LIN {X 0,Y 82.833,Z 534.203,A -85,B 0,C 180,E1 -27639.758,E2 -27639.758} C_VEL
LIN {X 0,Y 83.989,Z 533.266,A -85,B 0,C 180,E1 -27644.526,E2 -27644.526} C_VEL
LIN {X 0,Y 85.511,Z 531.952,A -85,B 0,C 180,E1 -27649.181,E2 -27649.181} C_VEL
LIN {X 0,Y 88.778,Z 529.155,A -85,B 0,C 180,E1 -27655.798,E2 -27655.798} C_VEL
LIN {X 0,Y 93.286,Z 525.282,A -85,B 0,C 180,E1 -27661.815,E2 -27661.815} C_VEL
LIN {X 0,Y 98.668,Z 520.245,A -85,B 0,C 180,E1 -27667.247,E2 -27667.247} C_VEL
LIN {X 0,Y 105.001,Z 513.4,A -85,B 0,C 180,E1 -27672.584,E2 -27672.584} C_VEL
LIN {X 0,Y 110.86,Z 506.1,A -85,B 0,C 180,E1 -27676.792,E2 -27676.792} C_VEL
LIN {X 0,Y 116.617,Z 498.037,A -85,B 0,C 180,E1 -27680.194,E2 -27680.194} C_VEL
LIN {X 0,Y 121.989,Z 489.202,A -85,B 0,C 180,E1 -27683.054,E2 -27683.054} C_VEL
LIN {X 0,Y 127.559,Z 478.2,A -85,B 0,C 180,E1 -27685.719,E2 -27685.719} C_VEL
LIN {X 0,Y 128.173,Z 476.919,A -85,B 0,C 180,E1 -27685.963,E2 -27685.963} C_VEL
LIN {X 0,Y 128.999,Z 471.512,A -85,B 0,C 180,E1 -27688.215,E2 -27688.215} C_VEL
LIN {X 0,Y 128.591,Z 466.823,A -85,B 0,C 180,E1 -27690.963,E2 -27690.963} C_VEL
LIN {X 0,Y 127.608,Z 461.168,A -85,B 0,C 180,E1 -27694.732,E2 -27694.732} C_VEL
LIN {X 0,Y 126.153,Z 455.519,A -85,B 0,C 180,E1 -27699.313,E2 -27699.313} C_VEL
LIN {X 0,Y 124.735,Z 451.921,A -85,B 0,C 180,E1 -27703.39,E2 -27703.39} C_VEL
LIN {X 0,Y 123.462,Z 448.563,A -85,B 0,C 180,E1 -27708.09,E2 -27708.09} C_VEL
LIN {X 0,Y 122.428,Z 445.351,A -85,B 0,C 180,E1 -27715.059,E2 -27715.059} C_VEL
LIN {X 0,Y 122.377,Z 444.889,A -85,B 0,C 180,E1 -27720.41,E2 -27720.41} C_VEL
LIN {X 0,Y 122.486,Z 446.263,A -85,B 0,C 180,E1 -27723.288,E2 -27723.288} C_VEL
LIN {X 0,Y 123.15,Z 449.904,A -85,B 0,C 180,E1 -27728.304,E2 -27728.304} C_VEL
LIN {X 0,Y 124.989,Z 457.619,A -85,B 0,C 180,E1 -27735.177,E2 -27735.177} C_VEL
LIN {X 0,Y 126.556,Z 464.817,A -85,B 0,C 180,E1 -27739.778,E2 -27739.778} C_VEL
LIN {X 0,Y 127.843,Z 470.42,A -85,B 0,C 180,E1 -27743.015,E2 -27743.015} C_VEL
LIN {X 0,Y 125.155,Z 484.311,A -85,B 0,C 180,E1 -27746.063,E2 -27746.063} C_VEL
LIN {X 0,Y 123.577,Z 490.066,A -85,B 0,C 180,E1 -27747.393,E2 -27747.393} C_VEL
LIN {X 0,Y 118.187,Z 501.884,A -85,B 0,C 180,E1 -27749.598,E2 -27749.598} C_VEL
LIN {X 0,Y 112.239,Z 512.594,A -85,B 0,C 180,E1 -27752.312,E2 -27752.312} C_VEL
LIN {X 0,Y 106.056,Z 522.326,A -85,B 0,C 180,E1 -27755.749,E2 -27755.749} C_VEL
LIN {X 0,Y 100.298,Z 530.329,A -85,B 0,C 180,E1 -27759.592,E2 -27759.592} C_VEL
LIN {X 0,Y 94.122,Z 538.214,A -85,B 0,C 180,E1 -27764.833,E2 -27764.833} C_VEL
LIN {X 0,Y 88.78,Z 544.608,A -85,B 0,C 180,E1 -27770.722,E2 -27770.722} C_VEL
LIN {X 0,Y 84.577,Z 549.746,A -85,B 0,C 180,E1 -27777.323,E2 -27777.323} C_VEL
LIN {X 0,Y 81.613,Z 553.757,A -85,B 0,C 180,E1 -27784.51,E2 -27784.51} C_VEL
LIN {X 0,Y 80.342,Z 555.873,A -85,B 0,C 180,E1 -27789.532,E2 -27789.532} C_VEL
LIN {X 0,Y 79.565,Z 557.948,A -85,B 0,C 180,E1 -27796.314,E2 -27796.314} C_VEL
LIN {X 0,Y 79.705,Z 559.51,A -85,B 0,C 180,E1 -27804.954,E2 -27804.954} C_VEL
LIN {X 0,Y 80.417,Z 559.877,A -85,B 0,C 180,E1 -27810.012,E2 -27810.012} C_VEL
LIN {X 0,Y 79.813,Z 559.509,A -85,B 0,C 180,E1 -27815.064,E2 -27815.064} C_VEL
LIN {X 0,Y 79.646,Z 558.723,A -85,B 0,C 180,E1 -27820.177,E2 -27820.177} C_VEL
LIN {X 0,Y 79.905,Z 557.516,A -85,B 0,C 180,E1 -27825.312,E2 -27825.312} C_VEL
LIN {X 0,Y 81.437,Z 554.888,A -85,B 0,C 180,E1 -27832.864,E2 -27832.864} C_VEL
LIN {X 0,Y 84.334,Z 551.27,A -85,B 0,C 180,E1 -27840.013,E2 -27840.013} C_VEL
LIN {X 0,Y 89.332,Z 545.786,A -85,B 0,C 180,E1 -27847.457,E2 -27847.457} C_VEL
LIN {X 0,Y 89.839,Z 545.307,A -85,B 0,C 180,E1 -27847.979,E2 -27847.979} C_VEL
LIN {X 0,Y 101.006,Z 544.866,A -85,B 0,C 180,E1 -27859.954,E2 -27859.954} C_VEL
LIN {X 0,Y 105.346,Z 544.467,A -85,B 0,C 180,E1 -27863.102,E2 -27863.102} C_VEL
LIN {X 0,Y 96.759,Z 538.849,A -85,B 0,C 180,E1 -27869.442,E2 -27869.442} C_VEL
LIN {X 0,Y 88.329,Z 530.261,A -85,B 0,C 180,E1 -27879.022,E2 -27879.022} C_VEL
LIN {X 0,Y 83.096,Z 520.814,A -85,B 0,C 180,E1 -27889.032,E2 -27889.032} C_VEL
LIN {X 0,Y 82.33,Z 518.793,A -85,B 0,C 180,E1 -27891.411,E2 -27891.411} C_VEL
LIN {X 0,Y 81.635,Z 518.051,A -85,B 0,C 180,E1 -27895.063,E2 -27895.063} C_VEL
LIN {X 0,Y 82.102,Z 516.286,A -85,B 0,C 180,E1 -27900.002,E2 -27900.002} C_VEL
LIN {X 0,Y 82.708,Z 514.93,A -85,B 0,C 180,E1 -27904.876,E2 -27904.876} C_VEL
LIN {X 0,Y 84.487,Z 513.029,A -85,B 0,C 180,E1 -27909.579,E2 -27909.579} C_VEL
LIN {X 0,Y 88.142,Z 510.312,A -85,B 0,C 180,E1 -27916.865,E2 -27916.865} C_VEL
LIN {X 0,Y 96.42,Z 505.521,A -85,B 0,C 180,E1 -27925.936,E2 -27925.936} C_VEL
LIN {X 0,Y 105.323,Z 501.018,A -85,B 0,C 180,E1 -27932.266,E2 -27932.266} C_VEL
LIN {X 0,Y 110.649,Z 498.102,A -85,B 0,C 180,E1 -27934.867,E2 -27934.867} C_VEL
LIN {X 0,Y 114.44,Z 496.301,A -85,B 0,C 180,E1 -27936.743,E2 -27936.743} C_VEL
LIN {X 0,Y 114.902,Z 496.45,A -85,B 0,C 180,E1 -27937.289,E2 -27937.289} C_VEL
LIN {X 0,Y 114.491,Z 497.858,A -85,B 0,C 180,E1 -27938.218,E2 -27938.218} C_VEL
LIN {X 0,Y 112.735,Z 500.446,A -85,B 0,C 180,E1 -27939.209,E2 -27939.209} C_VEL
LIN {X 0,Y 105.09,Z 508.492,A -85,B 0,C 180,E1 -27941.444,E2 -27941.444} C_VEL
LIN {X 0,Y 103.107,Z 510.663,A -85,B 0,C 180,E1 -27942.499,E2 -27942.499} C_VEL
LIN {X 0,Y 96.352,Z 518.081,A -85,B 0,C 180,E1 -27947.556,E2 -27947.556} C_VEL
LIN {X 0,Y 89.384,Z 524.598,A -85,B 0,C 180,E1 -27953.851,E2 -27953.851} C_VEL
LIN {X 0,Y 84.032,Z 528.908,A -85,B 0,C 180,E1 -27959.868,E2 -27959.868} C_VEL
LIN {X 0,Y 81.236,Z 531.13,A -85,B 0,C 180,E1 -27964.357,E2 -27964.357} C_VEL
LIN {X 0,Y 78.937,Z 532.932,A -85,B 0,C 180,E1 -27969.124,E2 -27969.124} C_VEL
LIN {X 0,Y 77.222,Z 534.283,A -85,B 0,C 180,E1 -27974.142,E2 -27974.142} C_VEL
LIN {X 0,Y 75.944,Z 535.235,A -85,B 0,C 180,E1 -27979.321,E2 -27979.321} C_VEL
LIN {X 0,Y 74.808,Z 536.056,A -85,B 0,C 180,E1 -27989.987,E2 -27989.987} C_VEL
LIN {X 0,Y 75.939,Z 535.278,A -85,B 0,C 180,E1 -28000.653,E2 -28000.653} C_VEL
LIN {X 0,Y 77.211,Z 534.343,A -85,B 0,C 180,E1 -28005.834,E2 -28005.834} C_VEL
LIN {X 0,Y 78.913,Z 533.029,A -85,B 0,C 180,E1 -28010.856,E2 -28010.856} C_VEL
LIN {X 0,Y 82.515,Z 530.23,A -85,B 0,C 180,E1 -28017.92,E2 -28017.92} C_VEL
LIN {X 0,Y 87.401,Z 526.356,A -85,B 0,C 180,E1 -28024.24,E2 -28024.24} C_VEL
LIN {X 0,Y 93.181,Z 521.318,A -85,B 0,C 180,E1 -28029.859,E2 -28029.859} C_VEL
LIN {X 0,Y 100.066,Z 514.349,A -85,B 0,C 180,E1 -28035.383,E2 -28035.383} C_VEL
LIN {X 0,Y 106.178,Z 507.169,A -85,B 0,C 180,E1 -28039.554,E2 -28039.554} C_VEL
LIN {X 0,Y 112.253,Z 499.104,A -85,B 0,C 180,E1 -28042.948,E2 -28042.948} C_VEL
LIN {X 0,Y 117.905,Z 490.264,A -85,B 0,C 180,E1 -28045.78,E2 -28045.78} C_VEL
LIN {X 0,Y 123.741,Z 479.256,A -85,B 0,C 180,E1 -28048.406,E2 -28048.406} C_VEL
LIN {X 0,Y 124.423,Z 476.66,A -85,B 0,C 180,E1 -28049.444,E2 -28049.444} C_VEL
LIN {X 0,Y 124.623,Z 473.65,A -85,B 0,C 180,E1 -28051.107,E2 -28051.107} C_VEL
LIN {X 0,Y 124.263,Z 468.236,A -85,B 0,C 180,E1 -28054.791,E2 -28054.791} C_VEL
LIN {X 0,Y 123.587,Z 463.882,A -85,B 0,C 180,E1 -28058.306,E2 -28058.306} C_VEL
LIN {X 0,Y 122.813,Z 460.538,A -85,B 0,C 180,E1 -28061.654,E2 -28061.654} C_VEL
LIN {X 0,Y 122.045,Z 457.833,A -85,B 0,C 180,E1 -28064.98,E2 -28064.98} C_VEL
LIN {X 0,Y 121.32,Z 455.06,A -85,B 0,C 180,E1 -28069.147,E2 -28069.147} C_VEL
LIN {X 0,Y 120.821,Z 452.168,A -85,B 0,C 180,E1 -28075.829,E2 -28075.829} C_VEL
LIN {X 0,Y 120.907,Z 451.946,A -85,B 0,C 180,E1 -28080.415,E2 -28080.415} C_VEL
LIN {X 0,Y 120.951,Z 453.628,A -85,B 0,C 180,E1 -28083.538,E2 -28083.538} C_VEL
LIN {X 0,Y 121.287,Z 456.551,A -85,B 0,C 180,E1 -28087.385,E2 -28087.385} C_VEL
LIN {X 0,Y 122.41,Z 463.559,A -85,B 0,C 180,E1 -28093.804,E2 -28093.804} C_VEL
LIN {X 0,Y 123.355,Z 470.169,A -85,B 0,C 180,E1 -28098.216,E2 -28098.216} C_VEL
LIN {X 0,Y 124.012,Z 474.29,A -85,B 0,C 180,E1 -28100.744,E2 -28100.744} C_VEL
LIN {X 0,Y 120.797,Z 487.152,A -85,B 0,C 180,E1 -28103.743,E2 -28103.743} C_VEL
LIN {X 0,Y 119.72,Z 490.608,A -85,B 0,C 180,E1 -28104.596,E2 -28104.596} C_VEL
LIN {X 0,Y 114.096,Z 502.097,A -85,B 0,C 180,E1 -28106.748,E2 -28106.748} C_VEL
LIN {X 0,Y 107.866,Z 512.581,A -85,B 0,C 180,E1 -28109.393,E2 -28109.393} C_VEL
LIN {X 0,Y 101.992,Z 521.223,A -85,B 0,C 180,E1 -28112.443,E2 -28112.443} C_VEL
LIN {X 0,Y 94.669,Z 530.629,A -85,B 0,C 180,E1 -28117.074,E2 -28117.074} C_VEL
LIN {X 0,Y 88.108,Z 538.272,A -85,B 0,C 180,E1 -28122.471,E2 -28122.471} C_VEL
LIN {X 0,Y 81.565,Z 545.347,A -85,B 0,C 180,E1 -28129.758,E2 -28129.758} C_VEL
LIN {X 0,Y 77.256,Z 550.092,A -85,B 0,C 180,E1 -28136.935,E2 -28136.935} C_VEL
LIN {X 0,Y 74.301,Z 553.756,A -85,B 0,C 180,E1 -28144.823,E2 -28144.823} C_VEL
LIN {X 0,Y 72.561,Z 556.992,A -85,B 0,C 180,E1 -28155.588,E2 -28155.588} C_VEL
LIN {X 0,Y 72.613,Z 558.418,A -85,B 0,C 180,E1 -28164.459,E2 -28164.459} C_VEL
LIN {X 0,Y 73.336,Z 558.791,A -85,B 0,C 180,E1 -28170.013,E2 -28170.013} C_VEL
LIN {X 0,Y 72.723,Z 558.417,A -85,B 0,C 180,E1 -28175.559,E2 -28175.559} C_VEL
LIN {X 0,Y 72.838,Z 556.784,A -85,B 0,C 180,E1 -28185.237,E2 -28185.237} C_VEL
LIN {X 0,Y 74.855,Z 553.783,A -85,B 0,C 180,E1 -28195.006,E2 -28195.006} C_VEL
LIN {X 0,Y 78.192,Z 550.167,A -85,B 0,C 180,E1 -28202.649,E2 -28202.649} C_VEL
LIN {X 0,Y 82.904,Z 545.488,A -85,B 0,C 180,E1 -28209.493,E2 -28209.493} C_VEL
LIN {X 0,Y 86.143,Z 542.479,A -85,B 0,C 180,E1 -28212.874,E2 -28212.874} C_VEL
LIN {X 0,Y 95.313,Z 542.275,A -85,B 0,C 180,E1 -28221.931,E2 -28221.931} C_VEL
LIN {X 0,Y 96.208,Z 542.082,A -85,B 0,C 180,E1 -28222.918,E2 -28222.918} C_VEL
LIN {X 0,Y 86.816,Z 534.865,A -85,B 0,C 180,E1 -28230.943,E2 -28230.943} C_VEL
LIN {X 0,Y 79.323,Z 525.924,A -85,B 0,C 180,E1 -28241.268,E2 -28241.268} C_VEL
LIN {X 0,Y 77.81,Z 525.42,A -85,B 0,C 180,E1 -28244.28,E2 -28244.28} C_VEL
LIN {X 0,Y 78.095,Z 518.652,A -85,B 0,C 180,E1 -28268.064,E2 -28268.064} C_VEL
LIN {X 0,Y 84.543,Z 514.175,A -85,B 0,C 180,E1 -28280.207,E2 -28280.207} C_VEL
LIN {X 0,Y 93.773,Z 509.487,A -85,B 0,C 180,E1 -28289.156,E2 -28289.156} C_VEL
LIN {X 0,Y 100.734,Z 506.327,A -85,B 0,C 180,E1 -28293.929,E2 -28293.929} C_VEL
LIN {X 0,Y 108.996,Z 502.319,A -85,B 0,C 180,E1 -28297.779,E2 -28297.779} C_VEL
LIN {X 0,Y 108.664,Z 503.744,A -85,B 0,C 180,E1 -28299.081,E2 -28299.081} C_VEL
LIN {X 0,Y 103.107,Z 510.663,A -85,B 0,C 180,E1 -28302.499,E2 -28302.499} C_VEL
LIN {X 0,Y 99.686,Z 514.194,A -85,B 0,C 180,E1 -28304.373,E2 -28304.373} C_VEL
LIN {X 0,Y 92.734,Z 519.7,A -85,B 0,C 180,E1 -28307.025,E2 -28307.025} C_VEL
LIN {X 0,Y 85.549,Z 524.579,A -85,B 0,C 180,E1 -28310.147,E2 -28310.147} C_VEL
LIN {X 0,Y 81.903,Z 527.126,A -85,B 0,C 180,E1 -28312.816,E2 -28312.816} C_VEL
LIN {X 0,Y 76.426,Z 531.174,A -85,B 0,C 180,E1 -28319.603,E2 -28319.603} C_VEL
LIN {X 0,Y 72.42,Z 534.01,A -85,B 0,C 180,E1 -28327.145,E2 -28327.145} C_VEL
LIN {X 0,Y 70.492,Z 535.361,A -85,B 0,C 180,E1 -28332.583,E2 -28332.583} C_VEL
LIN {X 0,Y 69.07,Z 536.31,A -85,B 0,C 180,E1 -28338.244,E2 -28338.244} C_VEL
LIN {X 0,Y 67.791,Z 537.133,A -85,B 0,C 180,E1 -28349.986,E2 -28349.986} C_VEL
LIN {X 0,Y 69.064,Z 536.353,A -85,B 0,C 180,E1 -28361.728,E2 -28361.728} C_VEL
LIN {X 0,Y 70.48,Z 535.42,A -85,B 0,C 180,E1 -28367.392,E2 -28367.392} C_VEL
LIN {X 0,Y 72.395,Z 534.105,A -85,B 0,C 180,E1 -28372.834,E2 -28372.834} C_VEL
LIN {X 0,Y 76.384,Z 531.306,A -85,B 0,C 180,E1 -28380.386,E2 -28380.386} C_VEL
LIN {X 0,Y 81.695,Z 527.431,A -85,B 0,C 180,E1 -28387.011,E2 -28387.011} C_VEL
LIN {X 0,Y 87.911,Z 522.39,A -85,B 0,C 180,E1 -28392.79,E2 -28392.79} C_VEL
LIN {X 0,Y 95.307,Z 515.38,A -85,B 0,C 180,E1 -28398.418,E2 -28398.418} C_VEL
LIN {X 0,Y 101.77,Z 508.237,A -85,B 0,C 180,E1 -28402.558,E2 -28402.558} C_VEL
LIN {X 0,Y 108.174,Z 500.169,A -85,B 0,C 180,E1 -28405.913,E2 -28405.913} C_VEL
LIN {X 0,Y 114.108,Z 491.325,A -85,B 0,C 180,E1 -28408.694,E2 -28408.694} C_VEL
LIN {X 0,Y 119.658,Z 481.481,A -85,B 0,C 180,E1 -28410.991,E2 -28410.991} C_VEL
LIN {X 0,Y 120.04,Z 480.367,A -85,B 0,C 180,E1 -28411.408,E2 -28411.408} C_VEL
LIN {X 0,Y 120.371,Z 477.712,A -85,B 0,C 180,E1 -28413.038,E2 -28413.038} C_VEL
LIN {X 0,Y 120.385,Z 472.643,A -85,B 0,C 180,E1 -28416.792,E2 -28416.792} C_VEL
LIN {X 0,Y 119.988,Z 467.797,A -85,B 0,C 180,E1 -28421.206,E2 -28421.206} C_VEL
LIN {X 0,Y 119.505,Z 464.937,A -85,B 0,C 180,E1 -28424.653,E2 -28424.653} C_VEL
LIN {X 0,Y 118.986,Z 461.601,A -85,B 0,C 180,E1 -28429.792,E2 -28429.792} C_VEL
LIN {X 0,Y 118.898,Z 458.901,A -85,B 0,C 180,E1 -28436.61,E2 -28436.61} C_VEL
LIN {X 0,Y 119.048,Z 458.863,A -85,B 0,C 180,E1 -28440.421,E2 -28440.421} C_VEL
LIN {X 0,Y 119.078,Z 462.44,A -85,B 0,C 180,E1 -28445.821,E2 -28445.821} C_VEL
LIN {X 0,Y 119.52,Z 468.513,A -85,B 0,C 180,E1 -28451.739,E2 -28451.739} C_VEL
LIN {X 0,Y 119.946,Z 474.653,A -85,B 0,C 180,E1 -28456.158,E2 -28456.158} C_VEL
LIN {X 0,Y 120.179,Z 478.222,A -85,B 0,C 180,E1 -28458.407,E2 -28458.407} C_VEL
LIN {X 0,Y 116.094,Z 491.174,A -85,B 0,C 180,E1 -28461.605,E2 -28461.605} C_VEL
LIN {X 0,Y 110.309,Z 502.311,A -85,B 0,C 180,E1 -28463.697,E2 -28463.697} C_VEL
LIN {X 0,Y 103.803,Z 512.522,A -85,B 0,C 180,E1 -28466.245,E2 -28466.245} C_VEL
LIN {X 0,Y 96.945,Z 521.809,A -85,B 0,C 180,E1 -28469.572,E2 -28469.572} C_VEL
LIN {X 0,Y 89.242,Z 530.924,A -85,B 0,C 180,E1 -28474.241,E2 -28474.241} C_VEL
LIN {X 0,Y 82.254,Z 538.296,A -85,B 0,C 180,E1 -28479.757,E2 -28479.757} C_VEL
LIN {X 0,Y 76.15,Z 544.232,A -85,B 0,C 180,E1 -28486.215,E2 -28486.215} C_VEL
LIN {X 0,Y 71.271,Z 548.978,A -85,B 0,C 180,E1 -28493.743,E2 -28493.743} C_VEL
LIN {X 0,Y 67.8,Z 552.643,A -85,B 0,C 180,E1 -28502.212,E2 -28502.212} C_VEL
LIN {X 0,Y 65.571,Z 556.036,A -85,B 0,C 180,E1 -28514.708,E2 -28514.708} C_VEL
LIN {X 0,Y 65.526,Z 557.325,A -85,B 0,C 180,E1 -28523.858,E2 -28523.858} C_VEL
LIN {X 0,Y 66.253,Z 557.704,A -85,B 0,C 180,E1 -28530.015,E2 -28530.015} C_VEL
LIN {X 0,Y 65.636,Z 557.323,A -85,B 0,C 180,E1 -28536.162,E2 -28536.162} C_VEL
LIN {X 0,Y 65.857,Z 555.831,A -85,B 0,C 180,E1 -28546.177,E2 -28546.177} C_VEL
LIN {X 0,Y 68.404,Z 552.679,A -85,B 0,C 180,E1 -28557.554,E2 -28557.554} C_VEL
LIN {X 0,Y 72.253,Z 549.065,A -85,B 0,C 180,E1 -28565.721,E2 -28565.721} C_VEL
LIN {X 0,Y 77.499,Z 544.386,A -85,B 0,C 180,E1 -28572.87,E2 -28572.87} C_VEL
LIN {X 0,Y 83.213,Z 539.471,A -85,B 0,C 180,E1 -28578.113,E2 -28578.113} C_VEL
LIN {X 0,Y 83.961,Z 539.481,A -85,B 0,C 180,E1 -28578.898,E2 -28578.898} C_VEL
LIN {X 0,Y 86.779,Z 538.866,A -85,B 0,C 180,E1 -28583.025,E2 -28583.025} C_VEL
LIN {X 0,Y 79.255,Z 532.702,A -85,B 0,C 180,E1 -28590.082,E2 -28590.082} C_VEL
LIN {X 0,Y 77.027,Z 532.131,A -85,B 0,C 180,E1 -28592.86,E2 -28592.86} C_VEL
LIN {X 0,Y 70.369,Z 526.801,A -85,B 0,C 180,E1 -28614.27,E2 -28614.27} C_VEL
LIN {X 0,Y 73.252,Z 522.271,A -85,B 0,C 180,E1 -28631.065,E2 -28631.065} C_VEL
LIN {X 0,Y 82.345,Z 517.135,A -85,B 0,C 180,E1 -28645.263,E2 -28645.263} C_VEL
LIN {X 0,Y 98.671,Z 510.136,A -85,B 0,C 180,E1 -28657.201,E2 -28657.201} C_VEL
LIN {X 0,Y 100.317,Z 509.415,A -85,B 0,C 180,E1 -28657.976,E2 -28657.976} C_VEL
LIN {X 0,Y 98.411,Z 511.85,A -85,B 0,C 180,E1 -28659.561,E2 -28659.561} C_VEL
LIN {X 0,Y 91.299,Z 519.157,A -85,B 0,C 180,E1 -28664.585,E2 -28664.585} C_VEL
LIN {X 0,Y 83.818,Z 525.675,A -85,B 0,C 180,E1 -28671.02,E2 -28671.02} C_VEL
LIN {X 0,Y 81.903,Z 527.126,A -85,B 0,C 180,E1 -28672.816,E2 -28672.816} C_VEL
LIN {X 0,Y 78.412,Z 529.488,A -85,B 0,C 180,E1 -28675.791,E2 -28675.791} C_VEL
LIN {X 0,Y 71.806,Z 532.945,A -85,B 0,C 180,E1 -28680.787,E2 -28680.787} C_VEL
LIN {X 0,Y 65.833,Z 535.556,A -85,B 0,C 180,E1 -28686.962,E2 -28686.962} C_VEL
LIN {X 0,Y 63.52,Z 536.591,A -85,B 0,C 180,E1 -28691.669,E2 -28691.669} C_VEL
LIN {X 0,Y 61.144,Z 537.985,A -85,B 0,C 180,E1 -28703.384,E2 -28703.384} C_VEL
LIN {X 0,Y 60.774,Z 538.21,A -85,B 0,C 180,E1 -28709.984,E2 -28709.984} C_VEL
LIN {X 0,Y 62.216,Z 537.428,A -85,B 0,C 180,E1 -28723.041,E2 -28723.041} C_VEL
LIN {X 0,Y 63.812,Z 536.497,A -85,B 0,C 180,E1 -28729.277,E2 -28729.277} C_VEL
LIN {X 0,Y 65.98,Z 535.182,A -85,B 0,C 180,E1 -28735.201,E2 -28735.201} C_VEL
LIN {X 0,Y 70.418,Z 532.381,A -85,B 0,C 180,E1 -28743.275,E2 -28743.275} C_VEL
LIN {X 0,Y 76.209,Z 528.505,A -85,B 0,C 180,E1 -28750.188,E2 -28750.188} C_VEL
LIN {X 0,Y 82.901,Z 523.463,A -85,B 0,C 180,E1 -28756.085,E2 -28756.085} C_VEL
LIN {X 0,Y 90.088,Z 517.141,A -85,B 0,C 180,E1 -28761.253,E2 -28761.253} C_VEL
LIN {X 0,Y 97.666,Z 509.306,A -85,B 0,C 180,E1 -28765.827,E2 -28765.827} C_VEL
LIN {X 0,Y 104.404,Z 501.235,A -85,B 0,C 180,E1 -28769.102,E2 -28769.102} C_VEL
LIN {X 0,Y 110.624,Z 492.388,A -85,B 0,C 180,E1 -28771.801,E2 -28771.801} C_VEL
LIN {X 0,Y 115.596,Z 484.106,A -85,B 0,C 180,E1 -28773.687,E2 -28773.687} C_VEL
LIN {X 0,Y 116.05,Z 482.696,A -85,B 0,C 180,E1 -28774.358,E2 -28774.358} C_VEL
LIN {X 0,Y 116.5,Z 478.229,A -85,B 0,C 180,E1 -28777.847,E2 -28777.847} C_VEL
LIN {X 0,Y 116.581,Z 473.471,A -85,B 0,C 180,E1 -28782.456,E2 -28782.456} C_VEL
LIN {X 0,Y 116.406,Z 470.759,A -85,B 0,C 180,E1 -28786.024,E2 -28786.024} C_VEL
LIN {X 0,Y 116.332,Z 468.587,A -85,B 0,C 180,E1 -28789.557,E2 -28789.557} C_VEL
LIN {X 0,Y 116.58,Z 465.75,A -85,B 0,C 180,E1 -28796.542,E2 -28796.542} C_VEL
LIN {X 0,Y 116.788,Z 465.606,A -85,B 0,C 180,E1 -28799.999,E2 -28799.999} C_VEL
LIN {X 0,Y 116.633,Z 467.681,A -85,B 0,C 180,E1 -28803.453,E2 -28803.453} C_VEL
LIN {X 0,Y 116.441,Z 472.562,A -85,B 0,C 180,E1 -28808.677,E2 -28808.677} C_VEL
LIN {X 0,Y 116.481,Z 475.544,A -85,B 0,C 180,E1 -28811.307,E2 -28811.307} C_VEL
LIN {X 0,Y 116.408,Z 481.703,A -85,B 0,C 180,E1 -28815.761,E2 -28815.761} C_VEL
LIN {X 0,Y 112.784,Z 491.752,A -85,B 0,C 180,E1 -28818.416,E2 -28818.416} C_VEL
LIN {X 0,Y 108.375,Z 499.921,A -85,B 0,C 180,E1 -28819.926,E2 -28819.926} C_VEL
LIN {X 0,Y 101.567,Z 510.394,A -85,B 0,C 180,E1 -28822.285,E2 -28822.285} C_VEL
LIN {X 0,Y 95.001,Z 519.017,A -85,B 0,C 180,E1 -28825.038,E2 -28825.038} C_VEL
LIN {X 0,Y 87.092,Z 527.975,A -85,B 0,C 180,E1 -28829.13,E2 -28829.13} C_VEL
LIN {X 0,Y 79.014,Z 536.048,A -85,B 0,C 180,E1 -28834.662,E2 -28834.662} C_VEL
LIN {X 0,Y 73.201,Z 541.269,A -85,B 0,C 180,E1 -28839.841,E2 -28839.841} C_VEL
LIN {X 0,Y 67.641,Z 546.072,A -85,B 0,C 180,E1 -28846.658,E2 -28846.658} C_VEL
LIN {X 0,Y 62.646,Z 550.417,A -85,B 0,C 180,E1 -28855.9,E2 -28855.9} C_VEL
LIN {X 0,Y 60.48,Z 552.545,A -85,B 0,C 180,E1 -28862.321,E2 -28862.321} C_VEL
LIN {X 0,Y 58.573,Z 555.078,A -85,B 0,C 180,E1 -28873.711,E2 -28873.711} C_VEL
LIN {X 0,Y 58.443,Z 556.231,A -85,B 0,C 180,E1 -28883.11,E2 -28883.11} C_VEL
LIN {X 0,Y 59.169,Z 556.617,A -85,B 0,C 180,E1 -28890.017,E2 -28890.017} C_VEL
LIN {X 0,Y 58.559,Z 556.23,A -85,B 0,C 180,E1 -28896.91,E2 -28896.91} C_VEL
LIN {X 0,Y 58.912,Z 554.871,A -85,B 0,C 180,E1 -28907.385,E2 -28907.385} C_VEL
LIN {X 0,Y 62.135,Z 551.578,A -85,B 0,C 180,E1 -28920.614,E2 -28920.614} C_VEL
LIN {X 0,Y 66.552,Z 547.963,A -85,B 0,C 180,E1 -28929.335,E2 -28929.335} C_VEL
LIN {X 0,Y 73.249,Z 542.645,A -85,B 0,C 180,E1 -28937.532,E2 -28937.532} C_VEL
LIN {X 0,Y 76.668,Z 539.855,A -85,B 0,C 180,E1 -28940.555,E2 -28940.555} C_VEL
LIN {X 0,Y 78.011,Z 537.963,A -85,B 0,C 180,E1 -28942.781,E2 -28942.781} C_VEL
LIN {X 0,Y 65.096,Z 532.054,A -85,B 0,C 180,E1 -28967.533,E2 -28967.533} C_VEL
LIN {X 0,Y 67.36,Z 526.292,A -85,B 0,C 180,E1 -28992.047,E2 -28992.047} C_VEL
LIN {X 0,Y 76.977,Z 521.399,A -85,B 0,C 180,E1 -29007.164,E2 -29007.164} C_VEL
LIN {X 0,Y 91.291,Z 515.788,A -85,B 0,C 180,E1 -29018.018,E2 -29018.018} C_VEL
LIN {X 0,Y 85.337,Z 521.292,A -85,B 0,C 180,E1 -29022.15,E2 -29022.15} C_VEL
LIN {X 0,Y 78.486,Z 526.752,A -85,B 0,C 180,E1 -29027.795,E2 -29027.795} C_VEL
LIN {X 0,Y 72.239,Z 531.062,A -85,B 0,C 180,E1 -29034.271,E2 -29034.271} C_VEL
LIN {X 0,Y 68.886,Z 533.279,A -85,B 0,C 180,E1 -29039.313,E2 -29039.313} C_VEL
LIN {X 0,Y 66.008,Z 535.088,A -85,B 0,C 180,E1 -29044.777,E2 -29044.777} C_VEL
LIN {X 0,Y 63.52,Z 536.591,A -85,B 0,C 180,E1 -29051.669,E2 -29051.669} C_VEL
LIN {X 0,Y 61.538,Z 537.505,A -85,B 0,C 180,E1 -29056.717,E2 -29056.717} C_VEL
LIN {X 0,Y 57.434,Z 538.649,A -85,B 0,C 180,E1 -29065.364,E2 -29065.364} C_VEL
LIN {X 0,Y 54.933,Z 539.062,A -85,B 0,C 180,E1 -29073.076,E2 -29073.076} C_VEL
LIN {X 0,Y 54.475,Z 538.96,A -85,B 0,C 180,E1 -29079.272,E2 -29079.272} C_VEL
LIN {X 0,Y 54.718,Z 538.777,A -85,B 0,C 180,E1 -29081.326,E2 -29081.326} C_VEL
LIN {X 0,Y 57.229,Z 537.575,A -85,B 0,C 180,E1 -29091.599,E2 -29091.599} C_VEL
LIN {X 0,Y 59.702,Z 536.258,A -85,B 0,C 180,E1 -29098.072,E2 -29098.072} C_VEL
LIN {X 0,Y 64.665,Z 533.456,A -85,B 0,C 180,E1 -29106.69,E2 -29106.69} C_VEL
LIN {X 0,Y 70.993,Z 529.579,A -85,B 0,C 180,E1 -29113.845,E2 -29113.845} C_VEL
LIN {X 0,Y 78.199,Z 524.535,A -85,B 0,C 180,E1 -29119.79,E2 -29119.79} C_VEL
LIN {X 0,Y 85.876,Z 518.211,A -85,B 0,C 180,E1 -29124.902,E2 -29124.902} C_VEL
LIN {X 0,Y 93.903,Z 510.375,A -85,B 0,C 180,E1 -29129.372,E2 -29129.372} C_VEL
LIN {X 0,Y 100.98,Z 502.302,A -85,B 0,C 180,E1 -29132.522,E2 -29132.522} C_VEL
LIN {X 0,Y 107.487,Z 493.449,A -85,B 0,C 180,E1 -29135.098,E2 -29135.098} C_VEL
LIN {X 0,Y 111.888,Z 486.448,A -85,B 0,C 180,E1 -29136.64,E2 -29136.64} C_VEL
LIN {X 0,Y 112.698,Z 481.88,A -85,B 0,C 180,E1 -29140.687,E2 -29140.687} C_VEL
LIN {X 0,Y 113.024,Z 478.571,A -85,B 0,C 180,E1 -29144.393,E2 -29144.393} C_VEL
LIN {X 0,Y 113.205,Z 475.442,A -85,B 0,C 180,E1 -29149.265,E2 -29149.265} C_VEL
LIN {X 0,Y 113.439,Z 473.727,A -85,B 0,C 180,E1 -29152.881,E2 -29152.881} C_VEL
LIN {X 0,Y 113.826,Z 472.462,A -85,B 0,C 180,E1 -29156.459,E2 -29156.459} C_VEL
LIN {X 0,Y 114.09,Z 472.444,A -85,B 0,C 180,E1 -29159.999,E2 -29159.999} C_VEL
LIN {X 0,Y 113.71,Z 474.81,A -85,B 0,C 180,E1 -29163.542,E2 -29163.542} C_VEL
LIN {X 0,Y 113.257,Z 479.744,A -85,B 0,C 180,E1 -29168.743,E2 -29168.743} C_VEL
LIN {X 0,Y 112.712,Z 485.221,A -85,B 0,C 180,E1 -29173.062,E2 -29173.062} C_VEL
LIN {X 0,Y 110.986,Z 489.615,A -85,B 0,C 180,E1 -29174.346,E2 -29174.346} C_VEL
LIN {X 0,Y 108.9,Z 494.111,A -85,B 0,C 180,E1 -29175.479,E2 -29175.479} C_VEL
LIN {X 0,Y 102.19,Z 504.934,A -85,B 0,C 180,E1 -29177.437,E2 -29177.437} C_VEL
LIN {X 0,Y 95.19,Z 514.272,A -85,B 0,C 180,E1 -29179.754,E2 -29179.754} C_VEL
LIN {X 0,Y 86.251,Z 524.392,A -85,B 0,C 180,E1 -29183.585,E2 -29183.585} C_VEL
LIN {X 0,Y 77.787,Z 532.589,A -85,B 0,C 180,E1 -29188.278,E2 -29188.278} C_VEL
LIN {X 0,Y 71.253,Z 538.197,A -85,B 0,C 180,E1 -29193.057,E2 -29193.057} C_VEL
LIN {X 0,Y 64.203,Z 543.735,A -85,B 0,C 180,E1 -29200.006,E2 -29200.006} C_VEL
LIN {X 0,Y 58.399,Z 548.11,A -85,B 0,C 180,E1 -29208.579,E2 -29208.579} C_VEL
LIN {X 0,Y 54.142,Z 551.429,A -85,B 0,C 180,E1 -29218.742,E2 -29218.742} C_VEL
LIN {X 0,Y 51.604,Z 554.096,A -85,B 0,C 180,E1 -29232.417,E2 -29232.417} C_VEL
LIN {X 0,Y 51.369,Z 555.137,A -85,B 0,C 180,E1 -29242.156,E2 -29242.156} C_VEL
LIN {X 0,Y 52.051,Z 555.524,A -85,B 0,C 180,E1 -29250.019,E2 -29250.019} C_VEL
LIN {X 0,Y 51.491,Z 555.136,A -85,B 0,C 180,E1 -29257.864,E2 -29257.864} C_VEL
LIN {X 0,Y 51.994,Z 553.913,A -85,B 0,C 180,E1 -29268.89,E2 -29268.89} C_VEL
LIN {X 0,Y 56.087,Z 550.478,A -85,B 0,C 180,E1 -29284.345,E2 -29284.345} C_VEL
LIN {X 0,Y 61.165,Z 546.86,A -85,B 0,C 180,E1 -29293.604,E2 -29293.604} C_VEL
LIN {X 0,Y 68.125,Z 541.92,A -85,B 0,C 180,E1 -29301.479,E2 -29301.479} C_VEL
LIN {X 0,Y 69.412,Z 540.962,A -85,B 0,C 180,E1 -29302.594,E2 -29302.594} C_VEL
LIN {X 0,Y 67.164,Z 539.563,A -85,B 0,C 180,E1 -29306.861,E2 -29306.861} C_VEL
LIN {X 0,Y 58.185,Z 534.233,A -85,B 0,C 180,E1 -29333.065,E2 -29333.065} C_VEL
LIN {X 0,Y 61.303,Z 529.964,A -85,B 0,C 180,E1 -29353.258,E2 -29353.258} C_VEL
LIN {X 0,Y 71.504,Z 525.253,A -85,B 0,C 180,E1 -29369.438,E2 -29369.438} C_VEL
LIN {X 0,Y 81.182,Z 521.723,A -85,B 0,C 180,E1 -29377.303,E2 -29377.303} C_VEL
LIN {X 0,Y 80.798,Z 522.368,A -85,B 0,C 180,E1 -29378.46,E2 -29378.46} C_VEL
LIN {X 0,Y 73.438,Z 527.829,A -85,B 0,C 180,E1 -29384.113,E2 -29384.113} C_VEL
LIN {X 0,Y 66.669,Z 532.139,A -85,B 0,C 180,E1 -29390.747,E2 -29390.747} C_VEL
LIN {X 0,Y 62.963,Z 534.354,A -85,B 0,C 180,E1 -29396.057,E2 -29396.057} C_VEL
LIN {X 0,Y 59.733,Z 536.165,A -85,B 0,C 180,E1 -29401.907,E2 -29401.907} C_VEL
LIN {X 0,Y 56.828,Z 537.7,A -85,B 0,C 180,E1 -29409.669,E2 -29409.669} C_VEL
LIN {X 0,Y 54.18,Z 539.062,A -85,B 0,C 180,E1 -29422.529,E2 -29422.529} C_VEL
LIN {X 0,Y 53.757,Z 539.286,A -85,B 0,C 180,E1 -29429.982,E2 -29429.982} C_VEL
LIN {X 0,Y 54.718,Z 538.777,A -85,B 0,C 180,E1 -29441.326,E2 -29441.326} C_VEL
LIN {X 0,Y 55.215,Z 538.49,A -85,B 0,C 180,E1 -29445.384,E2 -29445.384} C_VEL
LIN {X 0,Y 55.541,Z 537.745,A -85,B 0,C 180,E1 -29453.54,E2 -29453.54} C_VEL
LIN {X 0,Y 56.995,Z 535.959,A -85,B 0,C 180,E1 -29465.5,E2 -29465.5} C_VEL
LIN {X 0,Y 59.765,Z 534.217,A -85,B 0,C 180,E1 -29471.463,E2 -29471.463} C_VEL
LIN {X 0,Y 60.32,Z 533.901,A -85,B 0,C 180,E1 -29472.185,E2 -29472.185} C_VEL
LIN {X 0,Y 68.695,Z 529.073,A -85,B 0,C 180,E1 -29480.089,E2 -29480.089} C_VEL
LIN {X 0,Y 76.585,Z 523.65,A -85,B 0,C 180,E1 -29485.656,E2 -29485.656} C_VEL
LIN {X 0,Y 84.823,Z 516.879,A -85,B 0,C 180,E1 -29490.425,E2 -29490.425} C_VEL
LIN {X 0,Y 93.489,Z 508.38,A -85,B 0,C 180,E1 -29494.408,E2 -29494.408} C_VEL
LIN {X 0,Y 100.922,Z 499.644,A -85,B 0,C 180,E1 -29497.297,E2 -29497.297} C_VEL
LIN {X 0,Y 107.482,Z 490.438,A -85,B 0,C 180,E1 -29499.449,E2 -29499.449} C_VEL
LIN {X 0,Y 108.121,Z 489.146,A -85,B 0,C 180,E1 -29500.045,E2 -29500.045} C_VEL
LIN {X 0,Y 108.962,Z 485.94,A -85,B 0,C 180,E1 -29503.319,E2 -29503.319} C_VEL
LIN {X 0,Y 109.509,Z 483.216,A -85,B 0,C 180,E1 -29507.018,E2 -29507.018} C_VEL
LIN {X 0,Y 110.146,Z 480.337,A -85,B 0,C 180,E1 -29512.667,E2 -29512.667} C_VEL
LIN {X 0,Y 110.694,Z 479.029,A -85,B 0,C 180,E1 -29516.358,E2 -29516.358} C_VEL
LIN {X 0,Y 110.962,Z 479.11,A -85,B 0,C 180,E1 -29519.999,E2 -29519.999} C_VEL
LIN {X 0,Y 110.327,Z 481.855,A -85,B 0,C 180,E1 -29523.651,E2 -29523.651} C_VEL
LIN {X 0,Y 109.705,Z 485.34,A -85,B 0,C 180,E1 -29527.36,E2 -29527.36} C_VEL
LIN {X 0,Y 109.1,Z 488.655,A -85,B 0,C 180,E1 -29530.202,E2 -29530.202} C_VEL
LIN {X 0,Y 108.155,Z 490.899,A -85,B 0,C 180,E1 -29531.003,E2 -29531.003} C_VEL
LIN {X 0,Y 105.809,Z 495.436,A -85,B 0,C 180,E1 -29532.123,E2 -29532.123} C_VEL
LIN {X 0,Y 98.643,Z 506.046,A -85,B 0,C 180,E1 -29533.942,E2 -29533.942} C_VEL
LIN {X 0,Y 91.406,Z 514.992,A -85,B 0,C 180,E1 -29536.077,E2 -29536.077} C_VEL
LIN {X 0,Y 83.606,Z 523.282,A -85,B 0,C 180,E1 -29539.01,E2 -29539.01} C_VEL
LIN {X 0,Y 74.624,Z 531.481,A -85,B 0,C 180,E1 -29543.365,E2 -29543.365} C_VEL
LIN {X 0,Y 67.551,Z 537.081,A -85,B 0,C 180,E1 -29547.863,E2 -29547.863} C_VEL
LIN {X 0,Y 59.787,Z 542.622,A -85,B 0,C 180,E1 -29554.659,E2 -29554.659} C_VEL
LIN {X 0,Y 53.155,Z 546.994,A -85,B 0,C 180,E1 -29563.376,E2 -29563.376} C_VEL
LIN {X 0,Y 48.093,Z 550.318,A -85,B 0,C 180,E1 -29574.256,E2 -29574.256} C_VEL
LIN {X 0,Y 44.664,Z 553.116,A -85,B 0,C 180,E1 -29590.744,E2 -29590.744} C_VEL
LIN {X 0,Y 44.288,Z 554.038,A -85,B 0,C 180,E1 -29600.892,E2 -29600.892} C_VEL
LIN {X 0,Y 44.931,Z 554.432,A -85,B 0,C 180,E1 -29610.022,E2 -29610.022} C_VEL
LIN {X 0,Y 44.439,Z 554.042,A -85,B 0,C 180,E1 -29619.122,E2 -29619.122} C_VEL
LIN {X 0,Y 45.122,Z 552.937,A -85,B 0,C 180,E1 -29630.858,E2 -29630.858} C_VEL
LIN {X 0,Y 48.741,Z 550.365,A -85,B 0,C 180,E1 -29645.246,E2 -29645.246} C_VEL
LIN {X 0,Y 54.048,Z 547.088,A -85,B 0,C 180,E1 -29655.683,E2 -29655.683} C_VEL
LIN {X 0,Y 60.919,Z 542.781,A -85,B 0,C 180,E1 -29663.884,E2 -29663.884} C_VEL
LIN {X 0,Y 61,Z 542.366,A -85,B 0,C 180,E1 -29664.829,E2 -29664.829} C_VEL
LIN {X 0,Y 51.823,Z 537.378,A -85,B 0,C 180,E1 -29692.209,E2 -29692.209} C_VEL
LIN {X 0,Y 55.086,Z 533.271,A -85,B 0,C 180,E1 -29714.786,E2 -29714.786} C_VEL
LIN {X 0,Y 67.6,Z 528.177,A -85,B 0,C 180,E1 -29733.7,E2 -29733.7} C_VEL
LIN {X 0,Y 70.89,Z 527.083,A -85,B 0,C 180,E1 -29736.504,E2 -29736.504} C_VEL
LIN {X 0,Y 71.264,Z 527.217,A -85,B 0,C 180,E1 -29737.891,E2 -29737.891} C_VEL
LIN {X 0,Y 63.826,Z 531.876,A -85,B 0,C 180,E1 -29744.277,E2 -29744.277} C_VEL
LIN {X 0,Y 59.231,Z 534.406,A -85,B 0,C 180,E1 -29749.241,E2 -29749.241} C_VEL
LIN {X 0,Y 53.642,Z 537.243,A -85,B 0,C 180,E1 -29758.374,E2 -29758.374} C_VEL
LIN {X 0,Y 50.782,Z 538.595,A -85,B 0,C 180,E1 -29765.448,E2 -29765.448} C_VEL
LIN {X 0,Y 48.661,Z 539.54,A -85,B 0,C 180,E1 -29773.19,E2 -29773.19} C_VEL
LIN {X 0,Y 46.74,Z 540.363,A -85,B 0,C 180,E1 -29789.979,E2 -29789.979} C_VEL
LIN {X 0,Y 48.652,Z 539.58,A -85,B 0,C 180,E1 -29806.771,E2 -29806.771} C_VEL
LIN {X 0,Y 50.764,Z 538.652,A -85,B 0,C 180,E1 -29814.519,E2 -29814.519} C_VEL
LIN {X 0,Y 53.609,Z 537.334,A -85,B 0,C 180,E1 -29821.605,E2 -29821.605} C_VEL
LIN {X 0,Y 60.32,Z 533.901,A -85,B 0,C 180,E1 -29832.185,E2 -29832.185} C_VEL
LIN {X 0,Y 63.433,Z 532.035,A -85,B 0,C 180,E1 -29836.494,E2 -29836.494} C_VEL
LIN {X 0,Y 67.951,Z 528.694,A -85,B 0,C 180,E1 -29843.62,E2 -29843.62} C_VEL
LIN {X 0,Y 73.059,Z 524.703,A -85,B 0,C 180,E1 -29849.728,E2 -29849.728} C_VEL
LIN {X 0,Y 76.874,Z 521.755,A -85,B 0,C 180,E1 -29852.386,E2 -29852.386} C_VEL
LIN {X 0,Y 84.573,Z 515.347,A -85,B 0,C 180,E1 -29856.047,E2 -29856.047} C_VEL
LIN {X 0,Y 92.222,Z 507.865,A -85,B 0,C 180,E1 -29858.96,E2 -29858.96} C_VEL
LIN {X 0,Y 100.773,Z 497.678,A -85,B 0,C 180,E1 -29861.81,E2 -29861.81} C_VEL
LIN {X 0,Y 103.968,Z 493.306,A -85,B 0,C 180,E1 -29862.672,E2 -29862.672} C_VEL
LIN {X 0,Y 104.487,Z 492.317,A -85,B 0,C 180,E1 -29863.388,E2 -29863.388} C_VEL
LIN {X 0,Y 105.36,Z 489.821,A -85,B 0,C 180,E1 -29866.497,E2 -29866.497} C_VEL
LIN {X 0,Y 105.765,Z 488.621,A -85,B 0,C 180,E1 -29868.5,E2 -29868.5} C_VEL
LIN {X 0,Y 106.403,Z 486.789,A -85,B 0,C 180,E1 -29872.407,E2 -29872.407} C_VEL
LIN {X 0,Y 107.191,Z 485.43,A -85,B 0,C 180,E1 -29876.239,E2 -29876.239} C_VEL
LIN {X 0,Y 107.388,Z 485.729,A -85,B 0,C 180,E1 -29879.999,E2 -29879.999} C_VEL
LIN {X 0,Y 106.449,Z 488.77,A -85,B 0,C 180,E1 -29883.784,E2 -29883.784} C_VEL
LIN {X 0,Y 105.691,Z 491.49,A -85,B 0,C 180,E1 -29886.586,E2 -29886.586} C_VEL
LIN {X 0,Y 105.322,Z 492.76,A -85,B 0,C 180,E1 -29887.668,E2 -29887.668} C_VEL
LIN {X 0,Y 103.317,Z 496.223,A -85,B 0,C 180,E1 -29888.499,E2 -29888.499} C_VEL
LIN {X 0,Y 95.493,Z 507.121,A -85,B 0,C 180,E1 -29890.212,E2 -29890.212} C_VEL
LIN {X 0,Y 88.031,Z 515.709,A -85,B 0,C 180,E1 -29892.104,E2 -29892.104} C_VEL
LIN {X 0,Y 79.926,Z 523.687,A -85,B 0,C 180,E1 -29894.758,E2 -29894.758} C_VEL
LIN {X 0,Y 70.507,Z 531.546,A -85,B 0,C 180,E1 -29898.794,E2 -29898.794} C_VEL
LIN {X 0,Y 61.566,Z 537.938,A -85,B 0,C 180,E1 -29904.087,E2 -29904.087} C_VEL
LIN {X 0,Y 53.362,Z 543.048,A -85,B 0,C 180,E1 -29911.083,E2 -29911.083} C_VEL
LIN {X 0,Y 46.242,Z 547.077,A -85,B 0,C 180,E1 -29920.578,E2 -29920.578} C_VEL
LIN {X 0,Y 42.412,Z 549.205,A -85,B 0,C 180,E1 -29928.516,E2 -29928.516} C_VEL
LIN {X 0,Y 39.513,Z 550.862,A -85,B 0,C 180,E1 -29937.782,E2 -29937.782} C_VEL
LIN {X 0,Y 37.78,Z 552.134,A -85,B 0,C 180,E1 -29948.442,E2 -29948.442} C_VEL
LIN {X 0,Y 37.223,Z 552.938,A -85,B 0,C 180,E1 -29959.144,E2 -29959.144} C_VEL
LIN {X 0,Y 37.805,Z 553.338,A -85,B 0,C 180,E1 -29970.026,E2 -29970.026} C_VEL
LIN {X 0,Y 37.415,Z 552.947,A -85,B 0,C 180,E1 -29980.853,E2 -29980.853} C_VEL
LIN {X 0,Y 40.002,Z 550.902,A -85,B 0,C 180,E1 -30001.836,E2 -30001.836} C_VEL
LIN {X 0,Y 44.943,Z 548.269,A -85,B 0,C 180,E1 -30014.753,E2 -30014.753} C_VEL
LIN {X 0,Y 51.731,Z 544.658,A -85,B 0,C 180,E1 -30024.632,E2 -30024.632} C_VEL
LIN {X 0,Y 51.884,Z 543.865,A -85,B 0,C 180,E1 -30027.196,E2 -30027.196} C_VEL
LIN {X 0,Y 45.315,Z 540.167,A -85,B 0,C 180,E1 -30051.081,E2 -30051.081} C_VEL
LIN {X 0,Y 51.946,Z 534.766,A -85,B 0,C 180,E1 -30083.95,E2 -30083.95} C_VEL
LIN {X 0,Y 60.554,Z 531.832,A -85,B 0,C 180,E1 -30095.475,E2 -30095.475} C_VEL
LIN {X 0,Y 61.688,Z 531.563,A -85,B 0,C 180,E1 -30097.084,E2 -30097.084} C_VEL
LIN {X 0,Y 54.109,Z 535.483,A -85,B 0,C 180,E1 -30104.383,E2 -30104.383} C_VEL
LIN {X 0,Y 47.808,Z 538.32,A -85,B 0,C 180,E1 -30113.959,E2 -30113.959} C_VEL
LIN {X 0,Y 44.489,Z 539.673,A -85,B 0,C 180,E1 -30121.687,E2 -30121.687} C_VEL
LIN {X 0,Y 41.993,Z 540.617,A -85,B 0,C 180,E1 -30130.42,E2 -30130.42} C_VEL
LIN {X 0,Y 39.723,Z 541.44,A -85,B 0,C 180,E1 -30149.975,E2 -30149.975} C_VEL
LIN {X 0,Y 41.982,Z 540.656,A -85,B 0,C 180,E1 -30169.536,E2 -30169.536} C_VEL
LIN {X 0,Y 44.469,Z 539.729,A -85,B 0,C 180,E1 -30178.277,E2 -30178.277} C_VEL
LIN {X 0,Y 47.77,Z 538.411,A -85,B 0,C 180,E1 -30186.023,E2 -30186.023} C_VEL
LIN {X 0,Y 55.226,Z 535.023,A -85,B 0,C 180,E1 -30196.966,E2 -30196.966} C_VEL
LIN {X 0,Y 64.417,Z 530.148,A -85,B 0,C 180,E1 -30204.883,E2 -30204.883} C_VEL
LIN {X 0,Y 72.858,Z 524.722,A -85,B 0,C 180,E1 -30210.215,E2 -30210.215} C_VEL
LIN {X 0,Y 76.874,Z 521.755,A -85,B 0,C 180,E1 -30212.386,E2 -30212.386} C_VEL
LIN {X 0,Y 80.669,Z 518.654,A -85,B 0,C 180,E1 -30214.788,E2 -30214.788} C_VEL
LIN {X 0,Y 86.061,Z 513.4,A -85,B 0,C 180,E1 -30219.225,E2 -30219.225} C_VEL
LIN {X 0,Y 91.397,Z 507.535,A -85,B 0,C 180,E1 -30223.067,E2 -30223.067} C_VEL
LIN {X 0,Y 94.918,Z 503.48,A -85,B 0,C 180,E1 -30224.58,E2 -30224.58} C_VEL
LIN {X 0,Y 100.683,Z 496.318,A -85,B 0,C 180,E1 -30226.116,E2 -30226.116} C_VEL
LIN {X 0,Y 101.31,Z 495.008,A -85,B 0,C 180,E1 -30227.987,E2 -30227.987} C_VEL
LIN {X 0,Y 102.289,Z 493.045,A -85,B 0,C 180,E1 -30232.1,E2 -30232.1} C_VEL
LIN {X 0,Y 103.264,Z 491.637,A -85,B 0,C 180,E1 -30236.096,E2 -30236.096} C_VEL
LIN {X 0,Y 103.34,Z 492.241,A -85,B 0,C 180,E1 -30239.998,E2 -30239.998} C_VEL
LIN {X 0,Y 102.047,Z 495.525,A -85,B 0,C 180,E1 -30243.948,E2 -30243.948} C_VEL
LIN {X 0,Y 101.047,Z 497.327,A -85,B 0,C 180,E1 -30244.76,E2 -30244.76} C_VEL
LIN {X 0,Y 93.625,Z 507.055,A -85,B 0,C 180,E1 -30246.06,E2 -30246.06} C_VEL
LIN {X 0,Y 85.112,Z 516.293,A -85,B 0,C 180,E1 -30247.837,E2 -30247.837} C_VEL
LIN {X 0,Y 75.565,Z 524.96,A -85,B 0,C 180,E1 -30250.488,E2 -30250.488} C_VEL
LIN {X 0,Y 65.295,Z 532.743,A -85,B 0,C 180,E1 -30254.435,E2 -30254.435} C_VEL
LIN {X 0,Y 55.892,Z 538.672,A -85,B 0,C 180,E1 -30259.484,E2 -30259.484} C_VEL
LIN {X 0,Y 47.146,Z 543.41,A -85,B 0,C 180,E1 -30266.615,E2 -30266.615} C_VEL
LIN {X 0,Y 39.479,Z 547.075,A -85,B 0,C 180,E1 -30276.808,E2 -30276.808} C_VEL
LIN {X 0,Y 33.602,Z 549.75,A -85,B 0,C 180,E1 -30291.175,E2 -30291.175} C_VEL
LIN {X 0,Y 30.964,Z 551.157,A -85,B 0,C 180,E1 -30305.203,E2 -30305.203} C_VEL
LIN {X 0,Y 30.204,Z 551.836,A -85,B 0,C 180,E1 -30316.578,E2 -30316.578} C_VEL
LIN {X 0,Y 30.67,Z 552.243,A -85,B 0,C 180,E1 -30330.032,E2 -30330.032} C_VEL
LIN {X 0,Y 30.421,Z 551.849,A -85,B 0,C 180,E1 -30343.39,E2 -30343.39} C_VEL
LIN {X 0,Y 34.116,Z 549.801,A -85,B 0,C 180,E1 -30368.206,E2 -30368.206} C_VEL
LIN {X 0,Y 40.16,Z 547.166,A -85,B 0,C 180,E1 -30381.99,E2 -30381.99} C_VEL
LIN {X 0,Y 42.587,Z 546.062,A -85,B 0,C 180,E1 -30385.64,E2 -30385.64} C_VEL
LIN {X 0,Y 43.417,Z 545.252,A -85,B 0,C 180,E1 -30388.697,E2 -30388.697} C_VEL
LIN {X 0,Y 39.859,Z 540.016,A -85,B 0,C 180,E1 -30430.16,E2 -30430.16} C_VEL
LIN {X 0,Y 51.141,Z 535.671,A -85,B 0,C 180,E1 -30455.122,E2 -30455.122} C_VEL
LIN {X 0,Y 50.465,Z 536.099,A -85,B 0,C 180,E1 -30457.512,E2 -30457.512} C_VEL
LIN {X 0,Y 42.334,Z 539.398,A -85,B 0,C 180,E1 -30468.361,E2 -30468.361} C_VEL
LIN {X 0,Y 38.45,Z 540.752,A -85,B 0,C 180,E1 -30476.717,E2 -30476.717} C_VEL
LIN {X 0,Y 35.459,Z 541.694,A -85,B 0,C 180,E1 -30486.617,E2 -30486.617} C_VEL
LIN {X 0,Y 32.705,Z 542.517,A -85,B 0,C 180,E1 -30509.97,E2 -30509.97} C_VEL
LIN {X 0,Y 35.445,Z 541.733,A -85,B 0,C 180,E1 -30533.333,E2 -30533.333} C_VEL
LIN {X 0,Y 38.427,Z 540.806,A -85,B 0,C 180,E1 -30543.245,E2 -30543.245} C_VEL
LIN {X 0,Y 42.294,Z 539.487,A -85,B 0,C 180,E1 -30551.625,E2 -30551.625} C_VEL
LIN {X 0,Y 49.409,Z 536.682,A -85,B 0,C 180,E1 -30561.441,E2 -30561.441} C_VEL
LIN {X 0,Y 57.684,Z 532.802,A -85,B 0,C 180,E1 -30568.489,E2 -30568.489} C_VEL
LIN {X 0,Y 66.581,Z 527.753,A -85,B 0,C 180,E1 -30573.76,E2 -30573.76} C_VEL
LIN {X 0,Y 75.754,Z 521.426,A -85,B 0,C 180,E1 -30578.047,E2 -30578.047} C_VEL
LIN {X 0,Y 85.132,Z 513.58,A -85,B 0,C 180,E1 -30581.649,E2 -30581.649} C_VEL
LIN {X 0,Y 93.164,Z 505.497,A -85,B 0,C 180,E1 -30584.073,E2 -30584.073} C_VEL
LIN {X 0,Y 94.918,Z 503.48,A -85,B 0,C 180,E1 -30584.58,E2 -30584.58} C_VEL
LIN {X 0,Y 95.916,Z 502.187,A -85,B 0,C 180,E1 -30585.452,E2 -30585.452} C_VEL
LIN {X 0,Y 96.386,Z 501.312,A -85,B 0,C 180,E1 -30587.163,E2 -30587.163} C_VEL
LIN {X 0,Y 96.944,Z 500.219,A -85,B 0,C 180,E1 -30589.963,E2 -30589.963} C_VEL
LIN {X 0,Y 97.305,Z 499.73,A -85,B 0,C 180,E1 -30590.509,E2 -30590.509} C_VEL
LIN {X 0,Y 98.946,Z 497.654,A -85,B 0,C 180,E1 -30595.925,E2 -30595.925} C_VEL
LIN {X 0,Y 98.771,Z 498.618,A -85,B 0,C 180,E1 -30599.998,E2 -30599.998} C_VEL
LIN {X 0,Y 98.387,Z 499.394,A -85,B 0,C 180,E1 -30600.967,E2 -30600.967} C_VEL
LIN {X 0,Y 89.65,Z 509.89,A -85,B 0,C 180,E1 -30602.136,E2 -30602.136} C_VEL
LIN {X 0,Y 80.964,Z 518.441,A -85,B 0,C 180,E1 -30603.612,E2 -30603.612} C_VEL
LIN {X 0,Y 70.649,Z 526.878,A -85,B 0,C 180,E1 -30606.003,E2 -30606.003} C_VEL
LIN {X 0,Y 60.518,Z 533.752,A -85,B 0,C 180,E1 -30609.319,E2 -30609.319} C_VEL
LIN {X 0,Y 50.669,Z 539.285,A -85,B 0,C 180,E1 -30613.935,E2 -30613.935} C_VEL
LIN {X 0,Y 40.942,Z 543.818,A -85,B 0,C 180,E1 -30621.195,E2 -30621.195} C_VEL
LIN {X 0,Y 32.955,Z 546.975,A -85,B 0,C 180,E1 -30631.515,E2 -30631.515} C_VEL
LIN {X 0,Y 28.313,Z 548.636,A -85,B 0,C 180,E1 -30641.922,E2 -30641.922} C_VEL
LIN {X 0,Y 24.371,Z 550.165,A -85,B 0,C 180,E1 -30659.884,E2 -30659.884} C_VEL
LIN {X 0,Y 23.527,Z 551.147,A -85,B 0,C 180,E1 -30690.042,E2 -30690.042} C_VEL
LIN {X 0,Y 23.508,Z 550.749,A -85,B 0,C 180,E1 -30707.439,E2 -30707.439} C_VEL
LIN {X 0,Y 28.821,Z 548.699,A -85,B 0,C 180,E1 -30737.066,E2 -30737.066} C_VEL
LIN {X 0,Y 33.526,Z 547.055,A -85,B 0,C 180,E1 -30747.034,E2 -30747.034} C_VEL
LIN {X 0,Y 34.59,Z 546.114,A -85,B 0,C 180,E1 -30752.171,E2 -30752.171} C_VEL
LIN {X 0,Y 35.973,Z 540.826,A -85,B 0,C 180,E1 -30803.005,E2 -30803.005} C_VEL
LIN {X 0,Y 41.01,Z 539.191,A -85,B 0,C 180,E1 -30813.721,E2 -30813.721} C_VEL
LIN {X 0,Y 39.486,Z 539.777,A -85,B 0,C 180,E1 -30818.253,E2 -30818.253} C_VEL
LIN {X 0,Y 32.806,Z 541.83,A -85,B 0,C 180,E1 -30829.97,E2 -30829.97} C_VEL
LIN {X 0,Y 29.149,Z 542.772,A -85,B 0,C 180,E1 -30841.132,E2 -30841.132} C_VEL
LIN {X 0,Y 25.704,Z 543.592,A -85,B 0,C 180,E1 -30869.962,E2 -30869.962} C_VEL
LIN {X 0,Y 29.132,Z 542.81,A -85,B 0,C 180,E1 -30898.809,E2 -30898.809} C_VEL
LIN {X 0,Y 32.779,Z 541.884,A -85,B 0,C 180,E1 -30909.992,E2 -30909.992} C_VEL
LIN {X 0,Y 37.339,Z 540.563,A -85,B 0,C 180,E1 -30918.799,E2 -30918.799} C_VEL
LIN {X 0,Y 45.367,Z 537.758,A -85,B 0,C 180,E1 -30928.39,E2 -30928.39} C_VEL
LIN {X 0,Y 54.346,Z 533.876,A -85,B 0,C 180,E1 -30934.81,E2 -30934.81} C_VEL
LIN {X 0,Y 63.79,Z 528.826,A -85,B 0,C 180,E1 -30939.422,E2 -30939.422} C_VEL
LIN {X 0,Y 73.42,Z 522.498,A -85,B 0,C 180,E1 -30943.133,E2 -30943.133} C_VEL
LIN {X 0,Y 83.19,Z 514.649,A -85,B 0,C 180,E1 -30946.241,E2 -30946.241} C_VEL
LIN {X 0,Y 91.491,Z 506.561,A -85,B 0,C 180,E1 -30948.293,E2 -30948.293} C_VEL
LIN {X 0,Y 96.46,Z 500.852,A -85,B 0,C 180,E1 -30949.503,E2 -30949.503} C_VEL
LIN {X 0,Y 97.305,Z 499.73,A -85,B 0,C 180,E1 -30950.509,E2 -30950.509} C_VEL
LIN {X 0,Y 97.488,Z 499.455,A -85,B 0,C 180,E1 -30951.451,E2 -30951.451} C_VEL
LIN {X 0,Y 96.655,Z 500.451,A -85,B 0,C 180,E1 -30953.008,E2 -30953.008} C_VEL
LIN {X 0,Y 94.197,Z 503.466,A -85,B 0,C 180,E1 -30954.838,E2 -30954.838} C_VEL
LIN {X 0,Y 91.945,Z 506.075,A -85,B 0,C 180,E1 -30955.812,E2 -30955.812} C_VEL
LIN {X 0,Y 85.11,Z 513.324,A -85,B 0,C 180,E1 -30957.587,E2 -30957.587} C_VEL
LIN {X 0,Y 77.688,Z 520.043,A -85,B 0,C 180,E1 -30958.928,E2 -30958.928} C_VEL
LIN {X 0,Y 66.754,Z 528.22,A -85,B 0,C 180,E1 -30960.812,E2 -30960.812} C_VEL
LIN {X 0,Y 56.303,Z 534.602,A -85,B 0,C 180,E1 -30963.376,E2 -30963.376} C_VEL
LIN {X 0,Y 46.022,Z 539.722,A -85,B 0,C 180,E1 -30967.152,E2 -30967.152} C_VEL
LIN {X 0,Y 36.078,Z 543.732,A -85,B 0,C 180,E1 -30973.22,E2 -30973.22} C_VEL
LIN {X 0,Y 29.807,Z 545.86,A -85,B 0,C 180,E1 -30979.518,E2 -30979.518} C_VEL
LIN {X 0,Y 24.085,Z 547.526,A -85,B 0,C 180,E1 -30988.994,E2 -30988.994} C_VEL
LIN {X 0,Y 18.072,Z 549.18,A -85,B 0,C 180,E1 -31011.043,E2 -31011.043} C_VEL
LIN {X 0,Y 16.377,Z 550.05,A -85,B 0,C 180,E1 -31050.06,E2 -31050.06} C_VEL
LIN {X 0,Y 16.813,Z 549.65,A -85,B 0,C 180,E1 -31074.773,E2 -31074.773} C_VEL
LIN {X 0,Y 24.501,Z 547.597,A -85,B 0,C 180,E1 -31109.451,E2 -31109.451} C_VEL
LIN {X 0,Y 25.641,Z 547.287,A -85,B 0,C 180,E1 -31111.732,E2 -31111.732} C_VEL
LIN {X 0,Y 25.962,Z 546.614,A -85,B 0,C 180,E1 -31117.967,E2 -31117.967} C_VEL
LIN {X 0,Y 30.833,Z 542.194,A -85,B 0,C 180,E1 -31171.241,E2 -31171.241} C_VEL
LIN {X 0,Y 30.699,Z 542.193,A -85,B 0,C 180,E1 -31175.497,E2 -31175.497} C_VEL
LIN {X 0,Y 23.249,Z 543.849,A -85,B 0,C 180,E1 -31192.749,E2 -31192.749} C_VEL
LIN {X 0,Y 18.699,Z 544.667,A -85,B 0,C 180,E1 -31229.948,E2 -31229.948} C_VEL
LIN {X 0,Y 23.228,Z 543.887,A -85,B 0,C 180,E1 -31267.185,E2 -31267.185} C_VEL
LIN {X 0,Y 27.767,Z 542.961,A -85,B 0,C 180,E1 -31279.348,E2 -31279.348} C_VEL
LIN {X 0,Y 33.139,Z 541.639,A -85,B 0,C 180,E1 -31287.97,E2 -31287.97} C_VEL
LIN {X 0,Y 42.115,Z 538.833,A -85,B 0,C 180,E1 -31296.549,E2 -31296.549} C_VEL
LIN {X 0,Y 51.751,Z 534.95,A -85,B 0,C 180,E1 -31301.858,E2 -31301.858} C_VEL
LIN {X 0,Y 61.674,Z 529.899,A -85,B 0,C 180,E1 -31305.537,E2 -31305.537} C_VEL
LIN {X 0,Y 71.701,Z 523.567,A -85,B 0,C 180,E1 -31308.5,E2 -31308.5} C_VEL
LIN {X 0,Y 81.807,Z 515.717,A -85,B 0,C 180,E1 -31311.015,E2 -31311.015} C_VEL
LIN {X 0,Y 90.33,Z 507.627,A -85,B 0,C 180,E1 -31312.65,E2 -31312.65} C_VEL
LIN {X 0,Y 92.035,Z 505.775,A -85,B 0,C 180,E1 -31312.98,E2 -31312.98} C_VEL
LIN {X 0,Y 93.677,Z 504.002,A -85,B 0,C 180,E1 -31314.012,E2 -31314.012} C_VEL
LIN {X 0,Y 94.445,Z 503.3,A -85,B 0,C 180,E1 -31316.229,E2 -31316.229} C_VEL
LIN {X 0,Y 93.214,Z 504.861,A -85,B 0,C 180,E1 -31317.188,E2 -31317.188} C_VEL
LIN {X 0,Y 84.366,Z 514.09,A -85,B 0,C 180,E1 -31318.052,E2 -31318.052} C_VEL
LIN {X 0,Y 77.688,Z 520.043,A -85,B 0,C 180,E1 -31318.928,E2 -31318.928} C_VEL
LIN {X 0,Y 73.041,Z 523.683,A -85,B 0,C 180,E1 -31319.139,E2 -31319.139} C_VEL
LIN {X 0,Y 64.769,Z 529.008,A -85,B 0,C 180,E1 -31318.051,E2 -31318.051} C_VEL
LIN {X 0,Y 56.12,Z 533.713,A -85,B 0,C 180,E1 -31316.726,E2 -31316.726} C_VEL
LIN {X 0,Y 50.822,Z 536.29,A -85,B 0,C 180,E1 -31316.966,E2 -31316.966} C_VEL
LIN {X 0,Y 39.249,Z 541.189,A -85,B 0,C 180,E1 -31319.996,E2 -31319.996} C_VEL
LIN {X 0,Y 28.223,Z 544.747,A -85,B 0,C 180,E1 -31325.479,E2 -31325.479} C_VEL
LIN {X 0,Y 21.524,Z 546.412,A -85,B 0,C 180,E1 -31331.832,E2 -31331.832} C_VEL
LIN {X 0,Y 10.504,Z 548.529,A -85,B 0,C 180,E1 -31368.132,E2 -31368.132} C_VEL
LIN {X 0,Y 9.223,Z 548.952,A -85,B 0,C 180,E1 -31410.106,E2 -31410.106} C_VEL
LIN {X 0,Y 10.741,Z 548.551,A -85,B 0,C 180,E1 -31450.987,E2 -31450.987} C_VEL
LIN {X 0,Y 17.035,Z 547.469,A -85,B 0,C 180,E1 -31478.102,E2 -31478.102} C_VEL
LIN {X 0,Y 17.856,Z 546.764,A -85,B 0,C 180,E1 -31489.201,E2 -31489.201} C_VEL
LIN {X 0,Y 20.822,Z 544.653,A -85,B 0,C 180,E1 -31526.4,E2 -31526.4} C_VEL
LIN {X 0,Y 20.847,Z 544.518,A -85,B 0,C 180,E1 -31532.888,E2 -31532.888} C_VEL
LIN {X 0,Y 13.601,Z 545.521,A -85,B 0,C 180,E1 -31558.803,E2 -31558.803} C_VEL
LIN {X 0,Y 11.708,Z 545.74,A -85,B 0,C 180,E1 -31589.916,E2 -31589.916} C_VEL
LIN {X 0,Y 18.137,Z 544.964,A -85,B 0,C 180,E1 -31640.718,E2 -31640.718} C_VEL
LIN {X 0,Y 23.805,Z 544.035,A -85,B 0,C 180,E1 -31652.246,E2 -31652.246} C_VEL
LIN {X 0,Y 30.012,Z 542.716,A -85,B 0,C 180,E1 -31659.407,E2 -31659.407} C_VEL
LIN {X 0,Y 39.845,Z 539.909,A -85,B 0,C 180,E1 -31665.85,E2 -31665.85} C_VEL
LIN {X 0,Y 50.012,Z 536.024,A -85,B 0,C 180,E1 -31669.52,E2 -31669.52} C_VEL
LIN {X 0,Y 60.305,Z 530.972,A -85,B 0,C 180,E1 -31672.006,E2 -31672.006} C_VEL
LIN {X 0,Y 70.637,Z 524.638,A -85,B 0,C 180,E1 -31674.085,E2 -31674.085} C_VEL
LIN {X 0,Y 59.908,Z 531.528,A -85,B 0,C 180,E1 -31675.453,E2 -31675.453} C_VEL
LIN {X 0,Y 50.822,Z 536.29,A -85,B 0,C 180,E1 -31676.966,E2 -31676.966} C_VEL
LIN {X 0,Y 43.901,Z 539.292,A -85,B 0,C 180,E1 -31677.686,E2 -31677.686} C_VEL
LIN {X 0,Y 36.722,Z 541.75,A -85,B 0,C 180,E1 -31677.348,E2 -31677.348} C_VEL
LIN {X 0,Y 26.941,Z 544.299,A -85,B 0,C 180,E1 -31675.79,E2 -31675.79} C_VEL
LIN {X 0,Y 17.004,Z 546.155,A -85,B 0,C 180,E1 -31674.869,E2 -31674.869} C_VEL
LIN {X 0,Y 12.041,Z 546.825,A -85,B 0,C 180,E1 -31677.084,E2 -31677.084} C_VEL
LIN {X 0,Y 2.058,Z 547.852,A -85,B 0,C 180,E1 -31770.475,E2 -31770.475} C_VEL
LIN {X 0,Y 7.11,Z 547.454,A -85,B 0,C 180,E1 -31852.26,E2 -31852.26} C_VEL
LIN {X 0,Y 10.751,Z 547.053,A -85,B 0,C 180,E1 -31860.015,E2 -31860.015} C_VEL
LIN {X 0,Y 11.564,Z 546.499,A -85,B 0,C 180,E1 -31877.372,E2 -31877.372} C_VEL
LIN {X 0,Y 10.099,Z 546.47,A -85,B 0,C 180,E1 -31887.026,E2 -31887.026} C_VEL
LIN {X 0,Y 4.712,Z 546.813,A -85,B 0,C 180,E1 -31949.792,E2 -31949.792} C_VEL
LIN {X 0,Y 14.73,Z 546.041,A -85,B 0,C 180,E1 -32022.369,E2 -32022.369} C_VEL
LIN {X 0,Y 21.451,Z 545.115,A -85,B 0,C 180,E1 -32029.134,E2 -32029.134} C_VEL
LIN {X 0,Y 21.258,Z 545.299,A -85,B 0,C 180,E1 -32032.307,E2 -32032.307} C_VEL
LIN {X 0,Y 12.041,Z 546.825,A -85,B 0,C 180,E1 -32037.084,E2 -32037.084} C_VEL
LIN {X 0,Y 10.339,Z 548.808,A -85,B 0,C 180,E1 -32038.951,E2 -32038.951} C_VEL
LIN {X 0,Y 10.339,Z 600,A -85,B 0,C 180,E1 -32038.951,E2 -32038.951} C_VEL
LIN {X 0,Y 10.339,Z 600,A -85,B 0,C 180,E1 -32038.951,E2 -32038.951}

QRS_NEXT_CUT()

QRS_NEXT()
QRS_HOME()

END
